FUNCTION_BLOCK TFCiclo_Prelievo_Falda
VAR_INPUT
	Ciclo 		: POINTER TO Stato_Ciclo_Lavoro;
	Programma  : POINTER TO TFProgramma_Ciclo_Falda_Lastre;
	ModuleAX_X : POINTER TO TFModulePalletizer_Ax;
	ModuleAX_Y : POINTER TO TFModulePalletizer_Ax;
	ModuleAX_Z : POINTER TO TFModulePalletizer_Ax;
	ModuleAX_J : POINTER TO TFModulePalletizer_AxJ_Lastre;
	StartInterpolazioneAssi : POINTER TO BOOL;
	QuotaPassModePuntoIntermedio : ARRAY [1..3] OF REAL;
	ModulePinza : POINTER TO TFModulePalletizer_Pinza;
	AbilitazioneGlobalePassMode	: BOOL;
	InterrompiCiclo : BOOL;
	Abilita_Ciclo_Step : BOOL;
	Command_Step : BOOL;
	AbilitazioneAnticipoDinamicoMovimenti : bool;
END_VAR
VAR_OUTPUT
	STEPDone	: BOOL;
END_VAR
VAR
	ComandoInviatoTRIG : bool;
	StepInto: BOOL;
END_VAR

(* Set della variabile che mi permette di fare lo STEP nel ciclo *)
StepInto := (Abilita_Ciclo_Step AND Command_Step) OR NOT Abilita_Ciclo_Step;

(* Reset Anticipo Dinamico se non ho l'abilitazione *)
IF NOT AbilitazioneAnticipoDinamicoMovimenti  OR NOT HMI_DisabilitaAnticipiGLOBALE THEN
	QuotaAnticipoDinamicaX_Raggiunta := FALSE;
	QuotaAnticipoDinamicaY_Raggiunta := FALSE;
	QuotaAnticipoDinamicaZ_Raggiunta := FALSE;
END_IF

IF NOT InterrompiCiclo THEN
	IF Ciclo^.Stato = TERMINATO OR Ciclo^.Stato = ANNULLATO THEN
		Ciclo^.Passo := 0;
	ELSIF Ciclo^.Stato = INTERROTTO THEN
		Ciclo^.Passo := 999;
	END_IF
	Ciclo^.Stato := IN_ESECUZIONE;
	CASE Ciclo^.Passo OF
	(* Case 0 *)
			0:  Ciclo^.Stato := IN_ESECUZIONE;
				Ciclo^.Passo := 10;
				STEPDone := FALSE;
		
			(* Case 10 - Spengo aspirazione *)
			10:	IF ModulePinza^.CmdNext.Code = '' THEN
					IF (Abilita_Ciclo_Step AND Command_Step) OR NOT Abilita_Ciclo_Step THEN
						TFParametersArrayClear(ADR(ParametersArray));
						TFCommandSend(CmdUNLOAD,ParametersArray,ModulePinza^.Cmd);
						Ciclo^.Passo := 11;
						STEPDone := FALSE;
					END_IF
				END_IF
			(* Case 11 - Attesa aspirazione off*)
			11:
				IF TFStateCodeGet(ModulePinza^.State) = StateERROR  THEN
					Ciclo^.Passo := 0;	
					STEPDone := TRUE;
				ELSIF NOT TFStateCodeGet(ModulePinza^.State) = StateUNLOAD_RUN  THEN
					Ciclo^.Passo := 10;	
					STEPDone := TRUE;								
				ELSE
					IF TFStateCodeGet(ModulePinza^.State) = StateUNLOAD_END THEN
						Ciclo^.Passo := 20;
						STEPDone := TRUE;
					END_IF	
				END_IF;
				
			(* Case 20 - PROGRAMMA[0] ASSE Z -> TRASLAZIONE A QUOTA DI FUORI INGOMBRO *)	
			20:	Ciclo^.Stato := IN_ESECUZIONE;
				IF StepInto THEN
					TFParametersArrayClear(ADR(ParametersArray));
					Programma_Z[54].Stato := DA_ESEGUIRE;
					Programma_Z[54].InterpolaAsse := NO_INTERPOLAZIONE_ASSE;//FALSE;//NO_INTERPOLAZIONE_ASSE
					ProgrammaToModule_Z := Programma_Z[54];
					Ciclo^.Passo := 21;
					STEPDone := FALSE;
				END_IF
				
			(* Case 21 - Attesa completamento del comando MOVETOPOS o del raggiungimento quota di Pre-Movimento se abilitata la funzione*)
			21: 
				IF Programma_Z[54].Stato = TERMINATO OR 
					Asse_Z_InFinestraDiPassMode OR 
					QuotaAnticipoDinamicaZ_Raggiunta OR
					(ModuleAX_Z^.Ax^.Status.ActPosition >= QuotaFuoriIngombro_Z_AVUOTO-5) THEN
						Ciclo^.Passo := 22;
						STEPDone := TRUE;
				ELSIF Programma_Z[0].Stato = INTERROTTO THEN
					Ciclo^.Passo := 21;										
				END_IF
				
			(* Case 22 - Attesa completamento del comando MOVETOPOS o del raggiungimento quota di Pre-Movimento se abilitata la funzione *)
			22: IF Programma_Z[54].Stato = INTERROTTO THEN
					Ciclo^.Passo := 20;
				ELSE	
					Ciclo^.Passo := 23;
					STEPDone := TRUE;									
				END_IF
				
			(* Case 23 - Vado a quota di fuori ingombro colonne con Y *)
			23:
				IF Programma_Z[54].Stato = INTERROTTO THEN
					 Ciclo^.Passo := 20;										
				ELSE
					//IF FuoriIngombroYNecessario THEN
						IF StepInto THEN
							TFParametersArrayClear(ADR(ParametersArray));
							Programma_Y[56].Stato := DA_ESEGUIRE;
							Programma_Y[56].InterpolaAsse := NO_INTERPOLAZIONE_ASSE;
							ProgrammaToModule_Y := Programma_Y[56];
							Ciclo^.Passo := 24;
							STEPDone := FALSE;
						END_IF
					//ELSE
					//	Ciclo^.Passo := 24;
					//	STEPDone := FALSE;
					//END_IF
				END_IF
			
			(* Case 24 - *)
			24: IF Programma_Z[54].Stato = INTERROTTO OR
					Programma_Y[56].Stato = INTERROTTO THEN
						Ciclo^.Passo := 20;
				ELSIF Programma_Y[56].Stato = TERMINATO OR Asse_Y_InFinestraDiPassMode THEN// OR NOT FuoriIngombroYNecessario THEN	
					Ciclo^.Passo := 40;
					STEPDone := TRUE;									
				END_IF
				
			(* Case 40 - PROGRAMMA[] ASSE Y -> TRASLAZIONE A QUOTA DI PRELIEVO FALDA  *)	
			40:	
				IF Programma_Z[54].Stato = INTERROTTO OR 
					Programma_Y[56].Stato = INTERROTTO THEN
						Ciclo_Pelievo_Falda.Passo := 20;										
				ELSE
					IF StepInto THEN
						TFParametersArrayClear(ADR(ParametersArray));
						
						Programma_X[51].Stato := DA_ESEGUIRE;
						(*IF NOT Pinza_InIngombroColonne_Destinazione THEN
							Programma_Y[51].Stato := DA_ESEGUIRE;
							Programma_Y[54].InterpolaAsse := INTERPOLAZIONE_ASSE;//TRUE;//NO_INTERPOLAZIONE_ASSE
							ProgrammaToModule_Y := Programma_Y[51];
						END_IF*)
						Programma_J[10].Stato := DA_ESEGUIRE;
						Programma_K[51].Stato := DA_ESEGUIRE;
						
						Programma_X[51].InterpolaAsse := INTERPOLAZIONE_ASSE;//TRUE;//NO_INTERPOLAZIONE_ASSE
						//Programma_Y[54].InterpolaAsse := INTERPOLAZIONE_ASSE;//TRUE;//NO_INTERPOLAZIONE_ASSE
						Programma_J[10].InterpolaAsse := INTERPOLAZIONE_ASSE;//TRUE;//NO_INTERPOLAZIONE_ASSE
						Programma_K[51].InterpolaAsse := NO_INTERPOLAZIONE_ASSE;//FALSE;//NO_INTERPOLAZIONE_ASSE
						
						ProgrammaToModule_X := Programma_X[51];
						//ProgrammaToModule_Y := Programma_Y[51];
						ProgrammaToModule_J := Programma_J[10];
						ProgrammaToModule_K := Programma_K[51];
						
						ProgrammaToModule_Z.InterpolaAsse := NO_INTERPOLAZIONE_ASSE;//FALSE;//NO_INTERPOLAZIONE_ASSE
						
						StartInterpolazioneAssi^ := TRUE; //Abilito l'interpolazione degli assi
						
						TFCommandSend(CmdLOAD,ParametersArray,ModulePinza^.Cmd);
						
						Ciclo^.Passo := 41;
						STEPDone := FALSE;
					END_IF
				END_IF
				
			(* Case 41 - PROGRAMMA[51] ASSE Y -> TRASLAZIONE A QUOTA DI PRELIEVO FALDA  *)	
			41:	
				IF Programma_Z[54].Stato = INTERROTTO OR 
					Programma_Y[56].Stato = INTERROTTO OR 
					Programma_J[10].Stato = INTERROTTO OR 
					Programma_K[51].Stato = INTERROTTO OR 
					Programma_X[51].Stato = INTERROTTO THEN
					  Ciclo_Pelievo_Falda.Passo := 20;										
				ELSE
					STEPDone := TRUE;
					IF QuotaX_ConsensoRotazionePinza_Raggiunta OR NOT Pinza_InIngombroColonne_Destinazione THEN 
						IF StepInto THEN
							TFParametersArrayClear(ADR(ParametersArray));
							Programma_Y[51].Stato := DA_ESEGUIRE;
							Programma_Y[51].InterpolaAsse := NO_INTERPOLAZIONE_ASSE;
							ProgrammaToModule_Y := Programma_Y[51];
							
							Ciclo^.Passo := 42;
							STEPDone := FALSE;
						END_IF
					END_IF
				END_IF
					
			(* Case 42 -  Attesa completamento del comando MOVETOPOS o del raggiungimento quota di Pre-Movimento se abilitata la funzione *)
			42: 
				ComandoInviatoTRIG := FALSE;
				IF Programma_Z[54].Stato = INTERROTTO OR 
					Programma_Y[51].Stato = INTERROTTO OR  
					Programma_J[10].Stato = INTERROTTO OR 
					Programma_K[51].Stato = INTERROTTO OR 
					Programma_X[51].Stato = INTERROTTO THEN
						Ciclo^.Passo := 20;	
				ELSIF (Programma_X[51].Stato = TERMINATO OR Asse_X_InFinestraDiPassMode OR QuotaAnticipoDinamicaX_Raggiunta) AND 
					(Programma_Y[51].Stato = TERMINATO OR Asse_Y_InFinestraDiPassMode) AND
					(Programma_J[10].Stato = TERMINATO OR Asse_J_InFinestraDiPassMode) THEN
						Ciclo^.Passo := 80;
						STEPDone := TRUE;							
				END_IF
							
			(* Case 80 - PROGRAMMA[51] ASSE Z -> TRASLAZIONE A QUOTA AMMESSA IN VELOCE DI PRELIEVO FALDA  *)
			80:
				IF Programma_X[51].Stato = INTERROTTO THEN
					Ciclo^.Passo := 40;		//NON DOVREBBE MAI CAPITARE IN QUESTO PUNTO								
				ELSE
					IF StepInto THEN
						TFParametersArrayClear(ADR(ParametersArray));
						Programma_Z[51].Stato := DA_ESEGUIRE;
						Programma_Z[51].InterpolaAsse := NO_INTERPOLAZIONE_ASSE;//FALSE;//NO_INTERPOLAZIONE_ASSE
						ProgrammaToModule_Z := Programma_Z[51];
						Ciclo^.Passo := 81;
						STEPDone := FALSE;
					END_IF
				END_IF
			(* Case 81 -  Attesa completamento del comando MOVETOPOS o del raggiungimento quota di Pre-Movimento se abilitata la funzione *)
			81: 
				IF Programma_X[51].Stato = INTERROTTO OR 
				Programma_Z[51].Stato = INTERROTTO THEN
					Ciclo^.Passo := 40;									
				ELSE
					IF (Programma_Z[51].Stato = TERMINATO OR
					(ModuleAX_Z^.Ax^.Status.ActPosition <= Programma^.Quota_StartLenta_Prelievo_Falda_Z + 50 AND Programma_Z[51].Stato = IN_ESECUZIONE)) AND
					Programma_X[51].Stato = TERMINATO THEN	// controllo che la X sia in posizione corretta per poter iniziare la lenta senza collisioni
						Ciclo^.Passo := 100;
						STEPDone := TRUE;
					END_IF	
				END_IF
			
		 	(* Case 100 - PROGRAMMA[52] ASSE Z -> TRASLAZIONE IN LENTA A QUOTA DI PRELIEVO FALDA  *)
			100:
				IF Programma_Z[51].Stato = INTERROTTO THEN
					Ciclo^.Passo := 40; //NON DOVREBBE ACCADERE										
				ELSE
					IF StepInto THEN
						Programma_Z[52].Stato := DA_ESEGUIRE;
						Programma_Z[52].InterpolaAsse := NO_INTERPOLAZIONE_ASSE;//FALSE;//NO_INTERPOLAZIONE_ASSE
						ProgrammaToModule_Z := Programma_Z[52];
						Ciclo^.Passo := 101;
						STEPDone := FALSE;
					END_IF
				END_IF
				
			(* Case 101 -  Attesa completamento del comando MOVETOPOS o del raggiungimento quota di Pre-Movimento se abilitata la funzione *)
			101: 
				IF Programma_Z[52].Stato = INTERROTTO THEN
					Ciclo^.Passo := 20; //NON DOVREBBE ACCADERE										
				ELSE
					IF Programma_Z[52].Stato = TERMINATO THEN
						Ciclo^.Passo := 1000;
						STEPDone := TRUE;
					END_IF	
				END_IF
				
				(* Case 1000 *)
			1000:
				Ciclo^.Stato := TERMINATO;
				Ciclo^.Passo := 1000;
				
			(* Case 9999 - Ciclo NON annullato o NON terminato*)
			9999:
				Ciclo^.Stato := INTERROTTO;
				Ciclo^.Passo := 9999;
	ELSE						
		;
			
	END_CASE;
ELSE								//Se il ciclo deve essere interrotto, setto il suo nuovo stato
	Ciclo^.Stato := INTERROTTO;
END_IF

END_FUNCTION_BLOCK

(* stored: Version 1.1.0.1, ProductVersion 3.1.4024.11
   POU TFCiclo_Prelievo_Falda: Id {8f8f7049-ef68-4d30-83ed-2cb5a57f3cc8}, SpecialFunc None *)
